VISUALIZATION MainScreen  // 2x2
END_VISUALIZATION

(* stored: Version 1.1.0.1, ProductVersion 3.1.4024.15
   Visu MainScreen: Id {3c5eb390-ca10-415d-b24b-5a44a6258059} *)
